// TIA Portal V17 export
// export: Created 2024-06-14T09:52:50.1611908Z, ExportSetting WithDefaults, DisplayName Totally Integrated Automation Portal, DisplayVersion V17, DisplayName TIA Portal Openness, DisplayVersion V17, DisplayName TIA Portal Version Control Interface, DisplayVersion V17, DisplayName Simotion SCOUT TIA, DisplayVersion 5.4.3.0, DisplayName SINAMICS Startdrive Advanced, DisplayVersion V17 SP1 Update 1, DisplayName SINAMICS Startdrive G110M, G120, G120C, G120D, G120P, G115D, DisplayVersion V17 SP1 Update 1, DisplayName SINAMICS Startdrive G130, G150, S120, S150, SINAMICS MV, S210, DisplayVersion V17 SP1 Update 1, DisplayName STEP 7 Professional, DisplayVersion V17, DisplayName STEP 7 Safety, DisplayVersion V17, DisplayName WinCC Professional, DisplayVersion V17
DATA_BLOCK "FILLING_STATION5_DB"   // DB501
VERSION : 0.1
// stored: AutoNumber false, DBAccessibleFromOPCUA true, InstanceOfName FILLING_STATION5_FB, InstanceOfType FB
"FILLING_STATION5_FB"
   // VAR
   //    STATION5_S1 { S7_SetPoint := 'True'} : "LPG_FILLING_FB";
   //    STATION5_S2 { S7_SetPoint := 'True'} : "LPG_FILLING_FB";
   //    STATION5_S3 { S7_SetPoint := 'True'} : "LPG_FILLING_FB";
   //    STATION5_S4 { S7_SetPoint := 'True'} : "LPG_FILLING_FB";
   //    STATION5_S5 { S7_SetPoint := 'True'} : "LPG_FILLING_FB";
   //    STATION5_S6 { S7_SetPoint := 'True'} : "LPG_FILLING_FB";
   //    FILLING_STATION5 { S7_SetPoint := 'True'} : "FILLING_FB_L2";
   //    FILL_SEQ_STARTED_L2 { S7_SetPoint := 'True'} : Array[1..6] of Bool;
   //    FILLING_DONE_L2 : Array[1..6] of Bool;
   // END_VAR
BEGIN
END_DATA_BLOCK
